{attribute 'GeneratedUsingTerminal: EK1100-0000-0018'}
{attribute addProperty BoxType "EK1100-0000-0018"}
{attribute addProperty Id "EtcSlaveTerminalBaseInfoDataAT %I*InfoData_6F19DB2B2"}
{attribute addProperty CRC "2874840167"}
{attribute addProperty Size "2"}
TYPE EK1100_AB5A9467 EXTENDS EtcSlaveTerminalBase :
STRUCT
	{attribute addProperty Name "InfoData"}
	InfoData : InfoData_6F19DB2B;
END_STRUCT
END_TYPE

(* stored: Version 1.2.0.0, ProductVersion 3.1.4024.9
   DUT EK1100_AB5A9467: Id {79d68a1e-2c7e-46df-b5ce-1ac370e9ba23} *)
